Fanuc KAREL source: kf00114.KL

-- PROVISIONAL review KL for V770-1; original PC SHA256 3942bf497b8c738dcc0a10da4c0ba1203252529d6c9c9e04372d33a145cec109
-- Incomplete behavior may be omitted. Consult companion uncertainty JSON. Do not deploy.
PROGRAM KF00114
%NOLOCKGROUP
BEGIN
  -- UNRESOLVED_PC offsets 0-1; opcodes 7B
  -- UNRESOLVED_PC offsets 6-20; opcodes 2D,9D,52,23
  -- UNRESOLVED_PC offsets 25-29; opcodes 7F
  -- UNRESOLVED_PC offsets 34-44; opcodes 27,22,AA
  -- UNRESOLVED_PC offsets 49-53; opcodes 7F
END KF00114
